Staubli VAL3: goHome.dtx

public TrajBigBox pRunBigPt
  [0]
    bool bJtEnabCheck[6]
    bool bMoveJHomeJoint
    bool bPosEnabCheck[3]
    jointRx jToHome
    num nIndexGun
    num nRobCtrlAreaNum[6]
    num nRobCtrlHJtsNum[12]
public TrajJoint tTrajJoint
  [0]
    num nIndexFrame
    num nIndexTool
    string sID = "qwer"
    TrajJointItem tData[2]
      [0]
        jointRx jJoint = {j1=-15.581719, j2=14.249611, j3=85.047741, j5=80.702759, j6=3.379944}
        TrajectoryItem tSuper
          [0]
            string comment
            num distance
            InstrItem iInstr[3]
              [0]
                string sData
                string sType
              [1]
                string sData
                string sType
              [2]
                string sData
                string sType
            num moveType
            num nMoveId
            num nStop
            num nTcpAction
            num nTime
            mdesc nom_speed = {tmax=9999, rmax=9999, leave=30, reach=30}
            bool toStop
      [1]
        jointRx jJoint = {j1=21.410587, j2=14.249611, j3=85.047741, j5=80.702759, j6=3.379944}
        TrajectoryItem tSuper
          [0]
            string comment
            num distance
            InstrItem iInstr[3]
              [0]
                string sData
                string sType
              [1]
                string sData
                string sType
              [2]
                string sData
                string sType
            num moveType
            num nMoveId
            num nStop
            num nTcpAction
            num nTime
            mdesc nom_speed = {tmax=9999, rmax=9999, leave=30, reach=30}
            bool toStop
public TrajSmallBox pRunSmlPt
  [0]
    bool bMountOnWall
    bool bMoveJHomeJoint
    bool bReverse_Tool_Z
    string comment
    jointRx jToHome
    num nIndexGun
    num nKeySafeNum[6]
    num nRe_Tool_Z_Dits
    num nRe_Tool_Z_WrdX
    num nRe_Tool_Z_WrdY
    num nRe_Tool_Z_WrdZ
    num nToSafeFrmX
    num nToSafeFrmY
    num nToSafeFrmZ
    num nToSafePtType
    num nTolKeySafeNum[6]
    pointRx pPointRx
    pointRx pToSafePt
    num nToolType
public bool bWizard
public pointRx pPointRx = {x=539.985307, y=-152.401921, z=239.262224, rx=-0.000498, ry=179.999963, rz=-12.063425, fatherId=world[0]}
tool tTool = {fatherId=flange[0], ioLink=valve1}
num nSelected
string sEvent
string sList
bool bRefresh
bool bSelected
num nKey
num nIndex
num nView
string sMessage
public string sMenu[8]
num nRefresh
num nTime = 1
string sTitle
num nOldIndex
num nOldLine
bool bFaceA
public string sJointLimt[6]
public string sFrmRob[6]
bool bLocked
bool bFindInBox1
public string sHomingStatus
public string sBox1
public string sBox2
public mdesc mHomeSpd = {accel=10, vel=10, decel=10, blend=off}
num nSign
num nCurrentUseType
num nInWhichBox
num nShortP2PDists
num nShortP2PAngle
bool bSetMax
public Traies tTraies
  [0]
    frame fFrame
    num nIndexTool
    string sID
    num nIndexFrame
    TrajItem tData
      [0]
        TrajectoryItem tSuper
          [0]
            num distance
            num moveType
            num nTime
            num nStop
            num nTcpAction
            string comment
            bool toStop
            mdesc nom_speed = {vel=450, tmax=1000}
            InstrItem iInstr[3]
              [0]
                string sType
                string sData
              [1]
                string sType
                string sData
              [2]
                string sType
                string sData
            num nMoveId
        pointRx pPoint
        num nType
        pointRx pCircle
